FUNCTION_BLOCK Safety IMPLEMENTS I_Execute, I_Init
VAR
	_exe: Execute(THIS^);
	_init: Init(THIS^);	

	_bSafetyStopState: BOOL;
	_rtSafetyStop: R_TRIG;
	_ftSafetyStop: F_TRIG;
	
	_ett: EntityStart;
		_safetyStop: Signal;
	_ettEnd: EntityEnd;
END_VAR

(*
If registered, this method will be executed cyclically.
*)
METHOD Execute
VAR_INPUT
	nPhase	: INT;
END_VAR
VAR
	_safetyStopState: BoolArg(_bSafetyStopState);
END_VAR
_rtSafetyStop(CLk := _bSafetyStopState);
_ftSafetyStop(CLk := _bSafetyStopState);

IF _rtSafetyStop.Q OR _ftSafetyStop.Q THEN
	
	_safetyStop.Emit(_safetyStopState);
END_IF
END_METHOD

(*
If registered, this method will be executed upon startup.
*)
METHOD Init
VAR_INPUT
	nPhase	: INT;
END_VAR
VAR
	iEtt: I_Entity;
	iRec: I_Receiver;
END_VAR
WHILE IsOk(GetNextEntity(iEtt)) DO
	IF IsOk(GetReceiver(iEtt, '*._onSafetyStop.*', iRec)) THEN
		_safetyStop.Pair(iRec);
	END_IF
END_WHILE
END_METHOD

END_FUNCTION_BLOCK

(* stored: Version 1.1.0.1
   POU Safety: Id {d7d8a648-2a8b-4e3e-ae54-b27aadb17927}, SpecialFunc None
   Method Execute: Id {219d94b4-f298-481b-a6dd-5a1096aa2d8a}
   Method Init: Id {aad0f798-1e32-45e5-942d-4081f1f3400b} *)
